FUNCTION_BLOCK StructuredObject EXTENDS TcoCore.TcoObject

END_FUNCTION_BLOCK

(* stored: Version 1.1.0.1
   POU StructuredObject: Id {644525aa-e708-0d67-3a58-c68301fd1c62}, SpecialFunc None *)
